Staubli VAL3: IO.dtx

public dio diB_0_UPS = {link=BasicIO-1\%I0}
public dio diB_10 = {link=BasicIO-1\%I10}
public dio diB_11 = {link=BasicIO-1\%I11}
public dio diB_12 = {link=BasicIO-1\%I12}
public dio diB_13 = {link=BasicIO-1\%I13}
public dio diB_14 = {link=BasicIO-1\%I14}
public dio diB_15 = {link=BasicIO-1\%I15}
public dio diB_1_tableAlm = {link=BasicIO-1\%I1}
public dio diB_2_tableOn = {link=BasicIO-1\%I2}
public dio diB_3_toolAlm = {link=BasicIO-1\%I3}
public dio diB_4_tSpeedOk = {link=BasicIO-1\%I4}
public dio diB_5 = {link=BasicIO-1\%I5}
public dio diB_6 = {link=BasicIO-1\%I6}
public dio diB_7 = {link=BasicIO-1\%I7}
public dio diB_8 = {link=BasicIO-1\%I8}
public dio diB_9 = {link=BasicIO-1\%I9}
public dio doB_0_speed = {link=BasicIO-1\%Q0}
public dio doB_10_systeAlm = {link=BasicIO-1\%Q10}
public dio doB_11 = {link=BasicIO-1\%Q11}
public dio doB_12 = {link=BasicIO-1\%Q12}
public dio doB_13 = {link=BasicIO-1\%Q13}
public dio doB_14 = {link=BasicIO-1\%Q14}
public dio doB_15 = {link=BasicIO-1\%Q15}
public dio doB_1_speed = {link=BasicIO-1\%Q1}
public dio doB_2_speed = {link=BasicIO-1\%Q2}
public dio doB_3_speed = {link=BasicIO-1\%Q3}
public dio doB_4_speed = {link=BasicIO-1\%Q4}
public dio doB_5_speed = {link=BasicIO-1\%Q5}
public dio doB_6_toolPower = {link=BasicIO-1\%Q6}
public dio doB_7_toolOn = {link=BasicIO-1\%Q7}
public dio doB_8_toolOff = {link=BasicIO-1\%Q8}
public dio doB_9_tableOn = {link=BasicIO-1\%Q9}
mdesc mNomSpeed
public aio aRevolu = {link=ModbusSrv-0\Modbus-Word\Revolution}
public aio aRotation = {link=ModbusSrv-0\Modbus-Word\Rotation}
public aio aPressSet = {link=ModbusSrv-0\Modbus-Word\PressSet}
public aio aTableSpeed = {link=ModbusSrv-0\Modbus-Word\TableSpeed}
